    LAMP_C2_PTM_02(
    i_xExtILKOk:= F_Turbo_NC_NO_Valve_Logic_LL(
                    i_stTurbo:= LAMP_C2_PTM_02.iq_stPtm,
                    i_stISG:= LAMP_C2_GPI_01.PG,
                    i_stBSG:= LAMP_ROUGH_GPI_02.PG,
                    iq_stValve_NC:= LAMP_ROUGH_VRC_01.iq_stValve,
                    EcatBridge_Error_Present:= xEcatBridge_COM_ERROR,
//					ads_Error_Present:= (ITF_TMO_ROUGH1_VRC_01.bError OR ITF_TMO_ROUGH2_VRC_01.bError),
                    iq_stRoughRoughValve_NC_xOpnLS:= xTMO_ROUGH1_VRC_01_OPEN_LS,
                    x_onBeamline:= xOnBeamline),
//                    x_onBeamline:= True),
    iq_stPtm=> );

    LAMP_C2_PTM_03(
    i_xExtILKOk:= F_Turbo_NC_NO_Valve_Logic_LL(
                    i_stTurbo:= LAMP_C2_PTM_03.iq_stPtm,
                    i_stISG:= LAMP_C2_GPI_01.PG,
                    i_stBSG:= LAMP_ROUGH_GPI_02.PG,
                    iq_stValve_NC:= LAMP_ROUGH_VRC_01.iq_stValve,
                    EcatBridge_Error_Present:= xEcatBridge_COM_ERROR,
//					ads_Error_Present:= (ITF_TMO_ROUGH1_VRC_01.bError OR ITF_TMO_ROUGH2_VRC_01.bError),
                    iq_stRoughRoughValve_NC_xOpnLS:= xTMO_ROUGH1_VRC_01_OPEN_LS,
                    x_onBeamline:= xOnBeamline),
//                    x_onBeamline:= True),
    iq_stPtm=> );

    LAMP_C2_PTM_04(
    i_xExtILKOk:= F_Turbo_NC_NO_Valve_Logic_LL(
                    i_stTurbo:= LAMP_C2_PTM_04.iq_stPtm,
                    i_stISG:= LAMP_C2_GPI_01.PG,
                    i_stBSG:= LAMP_ROUGH_GPI_02.PG,
                    iq_stValve_NC:= LAMP_ROUGH_VRC_01.iq_stValve,
                    EcatBridge_Error_Present:= xEcatBridge_COM_ERROR,
//					ads_Error_Present:= (ITF_TMO_ROUGH1_VRC_01.bError OR ITF_TMO_ROUGH2_VRC_01.bError),
                    iq_stRoughRoughValve_NC_xOpnLS:= xTMO_ROUGH1_VRC_01_OPEN_LS,
                    x_onBeamline:= xOnBeamline),
//                    x_onBeamline:= True),
    iq_stPtm=> );


(*
    LAMP_CATCH_PTM_01(
    i_xExtILKOk:= F_Turbo_NC_NO_Valve_Logic(
                    i_stTurbo:= LAMP_CATCH_PTM_01.iq_stPtm,
                    i_stISG:= LAMP_C2_GPI_01.PG,
                    i_stBSG:= LAMP_ROUGH_GPI_02.PG,
                    iq_stValve_NO:= LAMP_ROUGH_VRC_02.iq_stValve,
                    iq_stValve_NC:= LAMP_ROUGH_VRC_01.iq_stValve,
                    iq_stValve_NC_second:= LAMP_ROUGH_VRC_03.iq_stValve,
                    EcatBridge_Error_Present:= xEcatBridge_COM_Error,
//					ads_Error_Present:= (ITF_TMO_ROUGH1_VRC_01.bError OR ITF_TMO_ROUGH2_VRC_01.bError),
                    iq_stRoughRoughValve_NC_xOpnLS:= xTMO_ROUGH1_VRC_01_OPEN_LS,
                    iq_stRoughRoughValve_NC_second_xOpenLS:=xTMO_ROUGH2_VRC_01_OPEN_LS,
                    x_onBeamline:= xOnBeamline),
    iq_stPtm=> );

    LAMP_CATCH_PTM_02(
    i_xExtILKOk:= F_Turbo_NC_NO_Valve_Logic(
                    i_stTurbo:= LAMP_CATCH_PTM_02.iq_stPtm,
                    i_stISG:= LAMP_C2_GPI_01.PG,
                    i_stBSG:= LAMP_ROUGH_GPI_02.PG,
                    iq_stValve_NO:= LAMP_ROUGH_VRC_02.iq_stValve,
                    iq_stValve_NC:= LAMP_ROUGH_VRC_01.iq_stValve,
                    iq_stValve_NC_second:= LAMP_ROUGH_VRC_03.iq_stValve,
                    EcatBridge_Error_Present:= xEcatBridge_COM_Error,
//					ads_Error_Present:= (ITF_TMO_ROUGH1_VRC_01.bError OR ITF_TMO_ROUGH2_VRC_01.bError),
                    iq_stRoughRoughValve_NC_xOpnLS:= xTMO_ROUGH1_VRC_01_OPEN_LS,
                    iq_stRoughRoughValve_NC_second_xOpenLS:=xTMO_ROUGH2_VRC_01_OPEN_LS,
                    x_onBeamline:= xOnBeamline),
    iq_stPtm=> );

    LAMP_GJ1_PTM_01(
    i_xExtILKOk:= F_Turbo_NC_NO_Valve_Logic(
                    i_stTurbo:= LAMP_GJ1_PTM_01.iq_stPtm,
                    i_stISG:= LAMP_GJ1_GPI_01.PG,
                    i_stBSG:= LAMP_ROUGH_GPI_04.PG,
                    iq_stValve_NO:= LAMP_ROUGH_VRC_02.iq_stValve,
                    iq_stValve_NC:= LAMP_ROUGH_VRC_03.iq_stValve,
                    iq_stValve_NC_second:= LAMP_ROUGH_VRC_01.iq_stValve,
                    EcatBridge_Error_Present:= xEcatBridge_COM_ERROR,
//					ads_Error_Present:= (ITF_TMO_ROUGH1_VRC_01.bError OR ITF_TMO_ROUGH2_VRC_01.bError),
                    iq_stRoughRoughValve_NC_xOpnLS:= xTMO_ROUGH2_VRC_01_OPEN_LS,
                    iq_stRoughRoughValve_NC_second_xOpenLS:=xTMO_ROUGH1_VRC_01_OPEN_LS,
                    x_onBeamline:= xOnBeamline),
    iq_stPtm=> );

    LAMP_GJ1_PTM_02(
    i_xExtILKOk:= F_Turbo_NC_NO_Valve_Logic(
                    i_stTurbo:= LAMP_GJ1_PTM_02.iq_stPtm,
                    i_stISG:= LAMP_GJ1_GPI_01.PG,
                    i_stBSG:= LAMP_ROUGH_GPI_04.PG,
                    iq_stValve_NO:= LAMP_ROUGH_VRC_02.iq_stValve,
                    iq_stValve_NC:= LAMP_ROUGH_VRC_03.iq_stValve,
                    iq_stValve_NC_second:= LAMP_ROUGH_VRC_01.iq_stValve,
                    EcatBridge_Error_Present:= xEcatBridge_COM_ERROR,
//					ads_Error_Present:= (ITF_TMO_ROUGH1_VRC_01.bError OR ITF_TMO_ROUGH2_VRC_01.bError),
                    iq_stRoughRoughValve_NC_xOpnLS:= xTMO_ROUGH2_VRC_01_OPEN_LS,
                    iq_stRoughRoughValve_NC_second_xOpenLS:=xTMO_ROUGH1_VRC_01_OPEN_LS,
                    x_onBeamline:= xOnBeamline),
    iq_stPtm=> );

    LAMP_GJ1_PTM_03(
    i_xExtILKOk:= F_Turbo_NC_NO_Valve_Logic(
                    i_stTurbo:= LAMP_GJ1_PTM_03.iq_stPtm,
                    i_stISG:= LAMP_GJ1_GPI_01.PG,
                    i_stBSG:= LAMP_ROUGH_GPI_04.PG,
                    iq_stValve_NO:= LAMP_ROUGH_VRC_02.iq_stValve,
                    iq_stValve_NC:= LAMP_ROUGH_VRC_03.iq_stValve,
                    iq_stValve_NC_second:= LAMP_ROUGH_VRC_01.iq_stValve,
                    EcatBridge_Error_Present:= xEcatBridge_COM_ERROR,
//					ads_Error_Present:= (ITF_TMO_ROUGH1_VRC_01.bError OR ITF_TMO_ROUGH2_VRC_01.bError),
                    iq_stRoughRoughValve_NC_xOpnLS:= xTMO_ROUGH2_VRC_01_OPEN_LS,
                    iq_stRoughRoughValve_NC_second_xOpenLS:=xTMO_ROUGH1_VRC_01_OPEN_LS,
                    x_onBeamline:= xOnBeamline),
    iq_stPtm=> );

    LAMP_GJ1_PTM_04(
    i_xExtILKOk:= F_Turbo_NC_NO_Valve_Logic(
                    i_stTurbo:= LAMP_GJ1_PTM_04.iq_stPtm,
                    i_stISG:= LAMP_GJ1_GPI_01.PG,
                    i_stBSG:= LAMP_ROUGH_GPI_04.PG,
                    iq_stValve_NO:= LAMP_ROUGH_VRC_02.iq_stValve,
                    iq_stValve_NC:= LAMP_ROUGH_VRC_03.iq_stValve,
                    iq_stValve_NC_second:= LAMP_ROUGH_VRC_01.iq_stValve,
                    EcatBridge_Error_Present:= xEcatBridge_COM_ERROR,
//					ads_Error_Present:= (ITF_TMO_ROUGH1_VRC_01.bError OR ITF_TMO_ROUGH2_VRC_01.bError),
                    iq_stRoughRoughValve_NC_xOpnLS:= xTMO_ROUGH2_VRC_01_OPEN_LS,
                    iq_stRoughRoughValve_NC_second_xOpenLS:=xTMO_ROUGH1_VRC_01_OPEN_LS,
                    x_onBeamline:= xOnBeamline),
    iq_stPtm=> );
*)

    LAMP_ROUGH_PTM_01(
    i_xExtILKOk:= F_Turbo_NC_NO_Valve_Logic(
                    i_stTurbo:= LAMP_ROUGH_PTM_01.iq_stPtm,
                    i_stISG:= LAMP_C2_GPI_01.PG,
                    i_stBSG:= LAMP_ROUGH_GPI_02.PG,
                    iq_stValve_NO:= LAMP_ROUGH_VRC_02.iq_stValve,
                    iq_stValve_NC:= LAMP_ROUGH_VRC_01.iq_stValve,
                    iq_stValve_NC_second:= LAMP_ROUGH_VRC_03.iq_stValve,
                    EcatBridge_Error_Present:= xEcatBridge_COM_ERROR,
//					ads_Error_Present:= (ITF_TMO_ROUGH1_VRC_01.bError OR ITF_TMO_ROUGH2_VRC_01.bError),
                    iq_stRoughRoughValve_NC_xOpnLS:= xTMO_ROUGH1_VRC_01_OPEN_LS,
                    iq_stRoughRoughValve_NC_second_xOpenLS:=xTMO_ROUGH2_VRC_01_OPEN_LS,
                    x_onBeamline:= xOnBeamline),
//                    x_onBeamline:= True),
    iq_stPtm=> );

(*
    KTOF_PTM_01(
    i_xExtILKOk:= F_Turbo_NC_NO_Valve_Logic(
                    i_stTurbo:= KTOF_PTM_01.iq_stPtm,
                    i_stISG:= LAMP_C2_GPI_01.PG,
                    i_stBSG:= LAMP_ROUGH_GPI_02.PG,
                    iq_stValve_NO:= LAMP_ROUGH_VRC_02.iq_stValve,
                    iq_stValve_NC:= LAMP_ROUGH_VRC_01.iq_stValve,
                    iq_stValve_NC_second:= LAMP_ROUGH_VRC_03.iq_stValve,
                    EcatBridge_Error_Present:= xEcatBridge_COM_ERROR,
//					ads_Error_Present:= (ITF_TMO_ROUGH1_VRC_01.bError OR ITF_TMO_ROUGH2_VRC_01.bError),
                    iq_stRoughRoughValve_NC_xOpnLS:= xTMO_ROUGH1_VRC_01_OPEN_LS,
                    iq_stRoughRoughValve_NC_second_xOpenLS:=xTMO_ROUGH2_VRC_01_OPEN_LS,
                    x_onBeamline:= xOnBeamline),
    iq_stPtm=> );
*)

(*Serial Communication*)
(*Assign adresses to the pfeiffer controllers connected to this serial terminal*)
st_Pfeiffer_CTRL_LAMP_C2_PTM_01[1].iSerialAddress :=1;
st_Pfeiffer_CTRL_LAMP_C2_PTM_01[1].xEnableComm := TRUE;
(* Instanitate the Function block for serial communication with Pfeiffer*)
fb_PfeifferCom_LAMP_C2_PTM_01(astPfeifferControl := st_Pfeiffer_CTRL_LAMP_C2_PTM_01,
                                 astPfeifferStatus:= st_Pfeiffer_RBK_LAMP_C2_PTM_01,
                              SerialRXBuffer:= SerialRXBuffer_LAMP_C2_PTM_01,
                              SerialTXBuffer:= SerialTXBuffer_LAMP_C2_PTM_01);
(* Copy Status Pv's into the PTM structure*)
LAMP_C2_PTM_01.M_Serial_IO(st_Pfeiffer_RBK:= st_Pfeiffer_RBK_LAMP_C2_PTM_01[1], st_Pfeiffer_CTRL:= st_Pfeiffer_CTRL_LAMP_C2_PTM_01[1]);

st_Pfeiffer_CTRL_LAMP_C2_PTM_02[1].iSerialAddress :=1;
st_Pfeiffer_CTRL_LAMP_C2_PTM_02[1].xEnableComm := TRUE;
fb_PfeifferCom_LAMP_C2_PTM_02(astPfeifferControl := st_Pfeiffer_CTRL_LAMP_C2_PTM_02,
                                 astPfeifferStatus:= st_Pfeiffer_RBK_LAMP_C2_PTM_02,
                              SerialRXBuffer:= SerialRXBuffer_LAMP_C2_PTM_02,
                              SerialTXBuffer:= SerialTXBuffer_LAMP_C2_PTM_02);
LAMP_C2_PTM_02.M_Serial_IO(st_Pfeiffer_RBK:= st_Pfeiffer_RBK_LAMP_C2_PTM_02[1], st_Pfeiffer_CTRL:= st_Pfeiffer_CTRL_LAMP_C2_PTM_02[1]);

st_Pfeiffer_CTRL_LAMP_C2_PTM_03[1].iSerialAddress :=1;
st_Pfeiffer_CTRL_LAMP_C2_PTM_03[1].xEnableComm := TRUE;
fb_PfeifferCom_LAMP_C2_PTM_03(astPfeifferControl := st_Pfeiffer_CTRL_LAMP_C2_PTM_03,
                                 astPfeifferStatus:= st_Pfeiffer_RBK_LAMP_C2_PTM_03,
                              SerialRXBuffer:= SerialRXBuffer_LAMP_C2_PTM_03,
                              SerialTXBuffer:= SerialTXBuffer_LAMP_C2_PTM_03);
LAMP_C2_PTM_03.M_Serial_IO(st_Pfeiffer_RBK:= st_Pfeiffer_RBK_LAMP_C2_PTM_03[1], st_Pfeiffer_CTRL:= st_Pfeiffer_CTRL_LAMP_C2_PTM_03[1]);

st_Pfeiffer_CTRL_LAMP_C2_PTM_04[1].iSerialAddress :=1;
st_Pfeiffer_CTRL_LAMP_C2_PTM_04[1].xEnableComm := TRUE;
fb_PfeifferCom_LAMP_C2_PTM_04(astPfeifferControl := st_Pfeiffer_CTRL_LAMP_C2_PTM_04,
                                 astPfeifferStatus:= st_Pfeiffer_RBK_LAMP_C2_PTM_04,
                              SerialRXBuffer:= SerialRXBuffer_LAMP_C2_PTM_04,
                              SerialTXBuffer:= SerialTXBuffer_LAMP_C2_PTM_04);

LAMP_C2_PTM_04.M_Serial_IO(st_Pfeiffer_RBK:= st_Pfeiffer_RBK_LAMP_C2_PTM_04[1], st_Pfeiffer_CTRL:= st_Pfeiffer_CTRL_LAMP_C2_PTM_04[1]);

(*
st_Pfeiffer_CTRL_LAMP_GJ1_PTM_01[1].iSerialAddress :=1;
st_Pfeiffer_CTRL_LAMP_GJ1_PTM_01[1].xEnableComm := TRUE;
fb_PfeifferCom_LAMP_GJ1_PTM_01(astPfeifferControl := st_Pfeiffer_CTRL_LAMP_GJ1_PTM_01,
                                 astPfeifferStatus:= st_Pfeiffer_RBK_LAMP_GJ1_PTM_01,
                              SerialRXBuffer:= SerialRXBuffer_LAMP_GJ1_PTM_01,
                              SerialTXBuffer:= SerialTXBuffer_LAMP_GJ1_PTM_01);
LAMP_GJ1_PTM_01.M_Serial_IO(st_Pfeiffer_RBK:= st_Pfeiffer_RBK_LAMP_GJ1_PTM_01[1], st_Pfeiffer_CTRL:= st_Pfeiffer_CTRL_LAMP_GJ1_PTM_01[1]);

st_Pfeiffer_CTRL_LAMP_GJ1_PTM_02[1].iSerialAddress :=1;
st_Pfeiffer_CTRL_LAMP_GJ1_PTM_02[1].xEnableComm := TRUE;
fb_PfeifferCom_LAMP_GJ1_PTM_02(astPfeifferControl := st_Pfeiffer_CTRL_LAMP_GJ1_PTM_02,
                                 astPfeifferStatus:= st_Pfeiffer_RBK_LAMP_GJ1_PTM_02,
                              SerialRXBuffer:= SerialRXBuffer_LAMP_GJ1_PTM_02,
                              SerialTXBuffer:= SerialTXBuffer_LAMP_GJ1_PTM_02);
LAMP_GJ1_PTM_02.M_Serial_IO(st_Pfeiffer_RBK:= st_Pfeiffer_RBK_LAMP_GJ1_PTM_02[1], st_Pfeiffer_CTRL:= st_Pfeiffer_CTRL_LAMP_GJ1_PTM_02[1]);

st_Pfeiffer_CTRL_LAMP_GJ1_PTM_03[1].iSerialAddress :=1;
st_Pfeiffer_CTRL_LAMP_GJ1_PTM_03[1].xEnableComm := TRUE;
fb_PfeifferCom_LAMP_GJ1_PTM_03(astPfeifferControl := st_Pfeiffer_CTRL_LAMP_GJ1_PTM_03,
                                 astPfeifferStatus:= st_Pfeiffer_RBK_LAMP_GJ1_PTM_03,
                              SerialRXBuffer:= SerialRXBuffer_LAMP_GJ1_PTM_03,
                              SerialTXBuffer:= SerialTXBuffer_LAMP_GJ1_PTM_03);
LAMP_GJ1_PTM_03.M_Serial_IO(st_Pfeiffer_RBK:= st_Pfeiffer_RBK_LAMP_GJ1_PTM_03[1], st_Pfeiffer_CTRL:= st_Pfeiffer_CTRL_LAMP_GJ1_PTM_03[1]);

st_Pfeiffer_CTRL_LAMP_GJ1_PTM_04[1].iSerialAddress :=1;
st_Pfeiffer_CTRL_LAMP_GJ1_PTM_04[1].xEnableComm := TRUE;
fb_PfeifferCom_LAMP_GJ1_PTM_04(astPfeifferControl := st_Pfeiffer_CTRL_LAMP_GJ1_PTM_04,
                                 astPfeifferStatus:= st_Pfeiffer_RBK_LAMP_GJ1_PTM_04,
                              SerialRXBuffer:= SerialRXBuffer_LAMP_GJ1_PTM_04,
                              SerialTXBuffer:= SerialTXBuffer_LAMP_GJ1_PTM_04);
LAMP_GJ1_PTM_04.M_Serial_IO(st_Pfeiffer_RBK:= st_Pfeiffer_RBK_LAMP_GJ1_PTM_04[1], st_Pfeiffer_CTRL:= st_Pfeiffer_CTRL_LAMP_GJ1_PTM_04[1]);
*)

st_Pfeiffer_CTRL_LAMP_ROUGH_PTM_01[1].iSerialAddress :=1;
st_Pfeiffer_CTRL_LAMP_ROUGH_PTM_01[1].xEnableComm := TRUE;
fb_PfeifferCom_LAMP_ROUGH_PTM_01(astPfeifferControl := st_Pfeiffer_CTRL_LAMP_ROUGH_PTM_01,
                                 astPfeifferStatus:= st_Pfeiffer_RBK_LAMP_ROUGH_PTM_01,
                              SerialRXBuffer:= SerialRXBuffer_LAMP_ROUGH_PTM_01,
                              SerialTXBuffer:= SerialTXBuffer_LAMP_ROUGH_PTM_01);
LAMP_ROUGH_PTM_01.M_Serial_IO(st_Pfeiffer_RBK:= st_Pfeiffer_RBK_LAMP_ROUGH_PTM_01[1], st_Pfeiffer_CTRL:= st_Pfeiffer_CTRL_LAMP_ROUGH_PTM_01[1]);

(*
st_Pfeiffer_CTRL_LAMP_C1_PTM_01[1].iSerialAddress :=1;
st_Pfeiffer_CTRL_LAMP_C1_PTM_01[1].xEnableComm := TRUE;
fb_PfeifferCom_LAMP_C1_PTM_01(astPfeifferControl := st_Pfeiffer_CTRL_LAMP_C1_PTM_01,
                                 astPfeifferStatus:= st_Pfeiffer_RBK_LAMP_C1_PTM_01,
                              SerialRXBuffer:= SerialRXBuffer_LAMP_C1_PTM_01,
                              SerialTXBuffer:= SerialTXBuffer_LAMP_C1_PTM_01);
LAMP_C1_PTM_01.M_Serial_IO(st_Pfeiffer_RBK:= st_Pfeiffer_RBK_LAMP_C1_PTM_01[1], st_Pfeiffer_CTRL:= st_Pfeiffer_CTRL_LAMP_C1_PTM_01[1]);

st_Pfeiffer_CTRL_LAMP_CATCH_PTM_01[1].iSerialAddress :=1;
st_Pfeiffer_CTRL_LAMP_CATCH_PTM_01[1].xEnableComm := TRUE;
fb_PfeifferCom_LAMP_CATCH_PTM_01(astPfeifferControl := st_Pfeiffer_CTRL_LAMP_CATCH_PTM_01,
                                 astPfeifferStatus:= st_Pfeiffer_RBK_LAMP_CATCH_PTM_01,
                              SerialRXBuffer:= SerialRXBuffer_LAMP_CATCH_PTM_01,
                              SerialTXBuffer:= SerialTXBuffer_LAMP_CATCH_PTM_01);
LAMP_CATCH_PTM_01.M_Serial_IO(st_Pfeiffer_RBK:= st_Pfeiffer_RBK_LAMP_CATCH_PTM_01[1], st_Pfeiffer_CTRL:= st_Pfeiffer_CTRL_LAMP_CATCH_PTM_01[1]);

st_Pfeiffer_CTRL_LAMP_CATCH_PTM_02[1].iSerialAddress :=1;
st_Pfeiffer_CTRL_LAMP_CATCH_PTM_02[1].xEnableComm := TRUE;
fb_PfeifferCom_LAMP_CATCH_PTM_02(astPfeifferControl := st_Pfeiffer_CTRL_LAMP_CATCH_PTM_02,
                                 astPfeifferStatus:= st_Pfeiffer_RBK_LAMP_CATCH_PTM_02,
                              SerialRXBuffer:= SerialRXBuffer_LAMP_CATCH_PTM_02,
                              SerialTXBuffer:= SerialTXBuffer_LAMP_CATCH_PTM_02);
LAMP_CATCH_PTM_02.M_Serial_IO(st_Pfeiffer_RBK:= st_Pfeiffer_RBK_LAMP_CATCH_PTM_02[1], st_Pfeiffer_CTRL:= st_Pfeiffer_CTRL_LAMP_CATCH_PTM_02[1]);

st_Pfeiffer_CTRL_KTOF_PTM_01[1].iSerialAddress :=1;
st_Pfeiffer_CTRL_KTOF_PTM_01[1].xEnableComm := TRUE;
fb_PfeifferCom_KTOF_PTM_01(astPfeifferControl := st_Pfeiffer_CTRL_KTOF_PTM_01,
                                 astPfeifferStatus:= st_Pfeiffer_RBK_KTOF_PTM_01,
                              SerialRXBuffer:= SerialRXBuffer_KTOF_PTM_01,
                              SerialTXBuffer:= SerialTXBuffer_KTOF_PTM_01);
//KTOF_PTM_01.M_Serial_IO(st_Pfeiffer_CTRL_KTOF_PTM_01[1],st_Pfeiffer_RBK_KTOF_PTM_01[1]);
KTOF_PTM_01.M_Serial_IO(st_Pfeiffer_RBK:= st_Pfeiffer_RBK_KTOF_PTM_01[1], st_Pfeiffer_CTRL:= st_Pfeiffer_CTRL_KTOF_PTM_01[1]);
*)

//Leybolds
fb_TD20Com_LAMP_GJ2_PTM_01(SerialRXBuffer:= SerialRXBuffer_LAMP_GJ2_PTM_01,
                           SerialTXBuffer:= SerialTXBuffer_LAMP_GJ2_PTM_01,
                           astTD20Status=> st_TD20_RBK_LAMP_GJ2_PTM_01);
LAMP_GJ2_PTM_01.M_Serial_IO(i_st_TD20_RBK:= st_TD20_RBK_LAMP_GJ2_PTM_01);

(*
fb_TD20Com_LAMP_GJ2_PTM_02(SerialRXBuffer:= SerialRXBuffer_LAMP_GJ2_PTM_02,
                           SerialTXBuffer:= SerialTXBuffer_LAMP_GJ2_PTM_02,
                           astTD20Status=> st_TD20_RBK_LAMP_GJ2_PTM_02);
LAMP_GJ2_PTM_02.M_Serial_IO(i_st_TD20_RBK:= st_TD20_RBK_LAMP_GJ2_PTM_02);

fb_TD20Com_LAMP_GJ2_PTM_03(SerialRXBuffer:= SerialRXBuffer_LAMP_GJ2_PTM_03,
                           SerialTXBuffer:= SerialTXBuffer_LAMP_GJ2_PTM_03,
                           astTD20Status=> st_TD20_RBK_LAMP_GJ2_PTM_03);
LAMP_GJ2_PTM_03.M_Serial_IO(i_st_TD20_RBK:= st_TD20_RBK_LAMP_GJ2_PTM_03);

fb_TD20Com_LAMP_GJ2_PTM_04(SerialRXBuffer:= SerialRXBuffer_LAMP_GJ2_PTM_04,
                           SerialTXBuffer:= SerialTXBuffer_LAMP_GJ2_PTM_04,
                           astTD20Status=> st_TD20_RBK_LAMP_GJ2_PTM_04);
LAMP_GJ2_PTM_04.M_Serial_IO(i_st_TD20_RBK:= st_TD20_RBK_LAMP_GJ2_PTM_04);
*)

(*Vacuum Gate Valve*)
    IF(xOnBeamline) THEN //If OnBeamline then stay open.
        LAMP_ROUGH_VRC_01.M_Set_OPN_SW(TRUE);
        LAMP_ROUGH_VRC_01(
        i_xExtILK_OK:= TRUE,
        i_xOverrideMode:= xSystemOverrideMode_LAMP,
        iq_stValve=> );
    ELSE
        LAMP_ROUGH_VRC_01(//LAMP:ROUGH:VRC:01 can open when the pressure across the valve is below 10 torr
        i_xExtILK_OK:= (ABS(LAMP_ROUGH_GPI_01.PG.rPRESS - LAMP_ROUGH_GPI_02.PG.rPRESS)<2000.0),
        i_xOverrideMode:= xSystemOverrideMode_LAMP,
        iq_stValve=> );
    END_IF
(*
    LAMP_ROUGH_VRC_02(//LAMP:ROUGH:VRC:02 closes when the pressure in the the C2, GJ1, and GJ2 chambers are all below 10 torr.
    i_xExtILK_OK:= NOT((LAMP_GJ1_GPI_01.PG.rPRESS >10.0) OR (LAMP_GJ2_GPI_01.PG.rPRESS > 10.0) OR (LAMP_C2_GPI_01.PG.rPRESS > 10.0)) ,
    i_xOverrideMode:= xSystemOverrideMode_LAMP,
    iq_stValve=> );
*)
    LAMP_ROUGH_VRC_02(//LAMP:ROUGH:VRC:02 close when the pressure in the C2, GJ1, GJ2 chambers are all below 10 torr.)
    i_xExtILK_OK:= NOT((LAMP_ROUGH_GPI_01.PG.rPRESS > 10.0 ) OR (LAMP_ROUGH_GPI_02.PG.rPRESS > 10.0) ),
    i_xOverrideMode:= xSystemOverrideMode_LAMP,
     iq_stValve=> );

    IF(xOnBeamline) THEN //If OnBeamline then stay open.
        LAMP_ROUGH_VRC_03.M_Set_OPN_SW(TRUE);
        LAMP_ROUGH_VRC_03(
        i_xExtILK_OK:= TRUE,
        i_xOverrideMode:= xSystemOverrideMode_LAMP,
        iq_stValve=> );

    ELSE
        LAMP_ROUGH_VRC_03(//LAMP:ROUGH:VRC:03 can open when the pressure across the valve is below 10 torr
        i_xExtILK_OK:= (ABS(LAMP_ROUGH_GPI_03.PG.rPRESS - LAMP_ROUGH_GPI_04.PG.rPRESS)<2000.0),
        i_xOverrideMode:= xSystemOverrideMode_LAMP,
        iq_stValve=> );
    END_IF

(*Update EtherCAT Bridge Outputs*)
xIP1_ROUGH_VRC_01_OPEN_LS := LAMP_ROUGH_VRC_01.M_IsOpen();
xIP1_ROUGH_VRC_02_OPEN_LS := LAMP_ROUGH_VRC_02.M_IsOpen();
xIP1_ROUGH_VRC_03_OPEN_LS := LAMP_ROUGH_VRC_03.M_IsOpen();
//xIP1_TURBO_FAULT AT %Q* : BOOL; already updated at turbo logic
xIP1_MAIN_xAT_VAC         := LAMP_C2_GCC_01.IG.xAT_VAC;
xIP1_MAIN_xPRESS_OK       := LAMP_C2_GCC_01.IG.xPRESS_OK;
rIP1_MAIN_rPRESS          := LAMP_C2_GCC_01.IG.rPRESS;
xIP1_HV_SAFETY_ENABLE     := xHighVoltageSafteyLoopEnable;


PRG_LAMP_GJ();

END_PROGRAM

// ---- POUs/DIAGNOSTICS.TcPOU
PROGRAM DIAGNOSTICS
VAR
    //Change the PLC String Name to the actual PLC NAME
    sPLCName :STRING := 'PLC-LAMP-VAC';
    //Link the sAMSNetID to the Etherat Master netID
    i_sAMSNetID AT %I*: AMSNETID;
    // DO NOT CHANGE
    sAMSNetID : STRING; //used for EPICS PV
    sLibVersion_LCLS_General : STRING;(* := stLibVersion_LCLS_General.sVersion*) ;
    fbEcatDiag:FB_EcatDiag;
    bAllSlaveStateGood : BOOL;
    bMasterStateGood :BOOL;
    iMasterState: WORD;
    sMasterState:STRING;
    nSlaveNumber : UINT;
    aiSlaveStates: ARRAY[1..256] OF BYTE;
    aEcSlaveInfo :  ARRAY[1..256] OF ST_EcDevice;
END_VAR

// Instaniating a call to the fbEcatDiag
fbEcatDiag(
    I_AMSNetId:=i_sAMSNetID ,
    i_xFirstPass:= _TaskInfo[1].FirstCycle,
    q_xAllSlaveStatesGood=> bAllSlaveStateGood ,
    q_anTermStates=> aiSlaveStates,
    q_xMasterStateGood=>bMasterStateGood ,
    q_nMasterState=> iMasterState,
    q_sMasterState=> sMasterState ,
    q_astEcConfSlaveInfo=> aEcSlaveInfo ,
    q_nSlaves=> nSlaveNumber);

END_PROGRAM

// ---- POUs/F_Turbo_NC_NO_Valve_Logic_LL.TcPOU
FUNCTION F_Turbo_NC_NO_Valve_Logic_LL : BOOL
VAR_INPUT
    i_stTurbo : ST_PTM; // Turbo Pump
    i_stISG : ST_VG; //Gauge measuring inlet Pressure e.g Pirani
    i_stBSG : ST_VG; //Gauge measureing backing pressure

    iq_stValve_NC : ST_VRC; //Normally Closed Valve directly sharing turbo pump vaccum volume.

    EcatBridge_Error_Present	:	BOOL; // Ecat Bridge Communication: Watchdog and Ecat Bridge Read Error Bit
//	ads_Error_Present     :      BOOL;  // ADS Communication: Watchdog and ADS Read Error Bit
    iq_stRoughRoughValve_NC_xOpnLS: BOOL; //Normally Closed Valve Downstream of iq_stValve_NC in Beamline Roughing Line.

    x_onBeamline :	BOOL; //Whether the  Turbopump/Endstation is mounted on the beamline or not.
END_VAR
VAR
END_VAR

IF (x_onBeamline) THEN
    F_Turbo_NC_NO_Valve_Logic_LL := (i_stISG.xPRESS_OK AND i_stISG.rPRESS < i_stTurbo.rInletPressureSP) AND
                                    (i_stBSG.xPRESS_OK AND i_stBSG.rPRESS < i_stTurbo.rBackingPressureSP) AND
                                 (iq_stValve_NC.i_xOpnLS AND iq_stRoughRoughValve_NC_xOpnLS) AND (NOT EcatBridge_Error_Present);
ELSE
    F_Turbo_NC_NO_Valve_Logic_LL := (i_stISG.xPRESS_OK AND i_stISG.rPRESS < i_stTurbo.rInletPressureSP) AND
                           (i_stBSG.xPRESS_OK AND i_stBSG.rPRESS < i_stTurbo.rBackingPressureSP) AND (iq_stValve_NC.i_xOpnLS);
END_IF

END_FUNCTION

// ---- POUs/F_Turbo_NC_NO_Valve_Logic.TcPOU
FUNCTION F_Turbo_NC_NO_Valve_Logic : BOOL
VAR_INPUT
    i_stTurbo : ST_PTM; // Turbo Pump
    i_stISG : ST_VG; //Gauge measuring inlet Pressure e.g Pirani
    i_stBSG : ST_VG; //Gauge measureing backing pressure
    iq_stValve_NO : ST_VRC_NO; //Normally Open Valve directly sharing turbo pump vaccum volume.
    iq_stValve_NC : ST_VRC; //Normally Closed Valve directly sharing turbo pump vaccum volume.
    iq_stValve_NC_second :	ST_VRC; //Normally Closed Valve on the other side of NO valve that also connects to roughing line.
    EcatBridge_Error_Present	:	BOOL; // Ecat Bridge Communication: Watchdog and Ecat Bridge Read Error Bit
//	ads_Error_Present     :      BOOL;  // ADS Communication: Watchdog and ADS Read Error Bit
    iq_stRoughRoughValve_NC_xOpnLS: BOOL; //Normally Closed Valve Downstream of iq_stValve_NC in Beamline Roughing Line.
    iq_stRoughRoughValve_NC_second_xOpenLS: BOOL; //Normally Closed Valve Downstream of iq_stValve_NC_second in Beamline Roughing Line.
    x_onBeamline :	BOOL; //Whether the  Turbopump/Endstation is mounted on the beamline or not.
END_VAR
VAR
END_VAR

IF (x_onBeamline) THEN
    F_Turbo_NC_NO_Valve_Logic := (i_stISG.xPRESS_OK AND i_stISG.rPRESS < i_stTurbo.rInletPressureSP) AND
                                    (i_stBSG.xPRESS_OK AND i_stBSG.rPRESS < i_stTurbo.rBackingPressureSP) AND
                                 ((iq_stValve_NC.i_xOpnLS AND iq_stRoughRoughValve_NC_xOpnLS) OR
                                 (iq_stValve_NO.i_xOpnLS AND (iq_stValve_NC_second.i_xOpnLS AND
                                 iq_stRoughRoughValve_NC_second_xOpenLS)))AND (NOT EcatBridge_Error_Present);
ELSE
    F_Turbo_NC_NO_Valve_Logic := (i_stISG.xPRESS_OK AND i_stISG.rPRESS < i_stTurbo.rInletPressureSP) AND
                           (i_stBSG.xPRESS_OK AND i_stBSG.rPRESS < i_stTurbo.rBackingPressureSP) AND
                            (iq_stValve_NC.i_xOpnLS OR(iq_stValve_NO.i_xOpnLS AND iq_stValve_NC_second.i_xOpnLS));
END_IF

END_FUNCTION

// ---- POUs/PRG_LAMP_GJ.TcPOU
PROGRAM PRG_LAMP_GJ
VAR
    {attribute 'pytmc' :=' pv:LAMP:GJ:VAC:OVERRIDE'}
    xSystemOverrideMode_LAMP_GJ : BOOL := FALSE;
	
	ROUGH_VRC_04_EXT_ILK_OK: BOOL;
	ROUGH_VRC_05_EXT_ILK_OK: BOOL;
	
	LAMP_GJ_VRC_01_OPN_OK: BOOL;
	LAMP_GJ_VRC_01_CLS_OK: BOOL;
	
	LAMP_GJ_01_EXT_INL_OK: BOOL;
	LAMP_GJ_PTM_01_PATH_1: BOOL;
	LAMP_GJ_PTM_01_PATH_2: BOOL;
	LAMP_GJ_PTM_01_PATH_3: BOOL;
	LAMP_GJ_VRC_02_EXT_ILK_OK: BOOL;
END_VAR

// VALVES

LAMP_GJ_VRC_01_OPN_OK:= (LAMP_C2_GCC_01.IG.rPRESS < 1E-6) 
						AND(LAMP_GJ_GCC_01.IG.rPRESS < 1E-6);
							
LAMP_GJ_VRC_01_CLS_OK:= (NOT LAMP_GJ_VRC_01_OPN_OK)
						AND (xLAMP_GJY_OUT AND NOT xEcat_External_Vac2Mot_device_not_connected);

LAMP_GJ_VRC_01(i_OPN_OK:=LAMP_GJ_VRC_01_OPN_OK,
            i_CLS_OK:=LAMP_GJ_VRC_01_CLS_OK,
            ibCntrlHold:=FALSE,
            i_xOverrideMode:=xSystemOverrideMode_LAMP_GJ,
            iq_stValve=>);
			
xLAMP_GJ_VRC_01_OPN_LS := LAMP_GJ_VRC_01.M_IsOpen(); // Send Valve Status to Motion


LAMP_GJ_VRC_02_EXT_ILK_OK := LAMP_ROUGH_VRC_02.M_IsClosed() AND LAMP_ROUGH_VRC_05.M_IsClosed();

LAMP_GJ_VRC_02(i_xExtILK_OK:=LAMP_GJ_VRC_02_EXT_ILK_OK,
            i_xOverrideMode:=xSystemOverrideMode_LAMP_GJ,
            iq_stValve=>);

			
ROUGH_VRC_04_EXT_ILK_OK := LAMP_ROUGH_VRC_05.M_IsClosed();
			
LAMP_ROUGH_VRC_04(i_stUSG:=LAMP_ROUGH_GPI_02.PG,
	i_stDSG:=LAMP_ROUGH_GPI_05.PG,
	i_xEPS_OK:=TRUE,
	i_xPMPS_OK:=TRUE,
	i_xExt_OK := ROUGH_VRC_04_EXT_ILK_OK,
	i_xOverrideMode:= xSystemOverrideMode_LAMP,
	io_fbFFHWO:= g_FastFaultOutput1 ,
	fbArbiter:= g_fbArbiter1,
	i_sDevName:= 'LAMP_ROUGH_VRC_04',
	iq_stValve=>);
	

ROUGH_VRC_05_EXT_ILK_OK := LAMP_ROUGH_VRC_04.M_IsClosed();	
	
LAMP_ROUGH_VRC_05(i_stUSG:=LAMP_ROUGH_GPI_04.PG,
	i_stDSG:=LAMP_ROUGH_GPI_05.PG,
	i_xEPS_OK:=TRUE,
	i_xPMPS_OK:=TRUE,
	i_xExt_OK := ROUGH_VRC_05_EXT_ILK_OK,
	i_xOverrideMode:= xSystemOverrideMode_LAMP,
	io_fbFFHWO:= g_FastFaultOutput1 ,
	fbArbiter:= g_fbArbiter1,
	i_sDevName:= 'LAMP_ROUGH_VRC_05',
	iq_stValve=>);
		
	
// GAUGES
LAMP_GJ_GPI_01.M_SetBits(30518);
LAMP_GJ_GPI_01();

LAMP_GJ_GCC_01.M_SetBits(30518);
LAMP_GJ_GCC_01(PG:=LAMP_GJ_GPI_01.PG, IG=>);

LAMP_ROUGH_GPI_05.M_SetBits(32767);
LAMP_ROUGH_GPI_05();


//PUMPS


LAMP_GJ_PTM_01_PATH_1:=(LAMP_ROUGH_VRC_04.M_IsOpen() 
						AND LAMP_ROUGH_VRC_01.M_IsOpen()
						AND (xTMO_ROUGH1_VRC_01_OPEN_LS OR NOT xOnBeamline));
						
LAMP_GJ_PTM_01_PATH_2:=(LAMP_ROUGH_VRC_05.M_IsOpen()
						AND LAMP_ROUGH_VRC_03.M_IsOpen()
						AND (xTMO_ROUGH2_VRC_01_OPEN_LS OR NOT xOnBeamline));
						
LAMP_GJ_PTM_01_PATH_3:=(LAMP_ROUGH_VRC_05.M_IsOpen()
						AND LAMP_ROUGH_VRC_02.M_IsOpen()
						AND LAMP_ROUGH_VRC_01.M_IsOpen()
						AND (xTMO_ROUGH1_VRC_01_OPEN_LS OR NOT xOnBeamline));

						
LAMP_GJ_01_EXT_INL_OK:= (NOT MAIN.xEcatBridge_COM_ERROR OR NOT xOnBeamline)
						AND (LAMP_GJ_PTM_01_PATH_1
							OR LAMP_GJ_PTM_01_PATH_2
							OR LAMP_GJ_PTM_01_PATH_3);

LAMP_GJ_PTM_01(i_xExtIlkOK:= LAMP_GJ_01_EXT_INL_OK, iq_stPTM=>);

st_Pfeiffer_CTRL_LAMP_GJ_PTM_01[1].iSerialAddress :=1;
st_Pfeiffer_CTRL_LAMP_GJ_PTM_01[1].xEnableComm := TRUE;
fb_PfeifferCom_LAMP_GJ_PTM_01(astPfeifferControl := st_Pfeiffer_CTRL_LAMP_GJ_PTM_01,
                                 astPfeifferStatus:= st_Pfeiffer_RBK_LAMP_GJ_PTM_01,
                              SerialRXBuffer:= SerialRXBuffer_LAMP_GJ_PTM_01,
                              SerialTXBuffer:= SerialTXBuffer_LAMP_GJ_PTM_01);
							  
LAMP_GJ_PTM_01.M_Serial_IO(st_Pfeiffer_RBK:= st_Pfeiffer_RBK_LAMP_GJ_PTM_01[1],
							st_Pfeiffer_CTRL:= st_Pfeiffer_CTRL_LAMP_GJ_PTM_01[1]);
					
IF NOT xTMO_ROUGH1_VRC_01_OPEN_LS THEN
	LAMP_C2_PTM_01.M_Run(False);
	LAMP_C2_PTM_02.M_Run(False);
	LAMP_C2_PTM_03.M_Run(False);
	LAMP_C2_PTM_04.M_Run(False);
	LAMP_GJ_PTM_01.M_Run(False);
END_IF

END_PROGRAM
